(* PLC project Water_Reserve_Control, Desconocido Sin nombre 1 *)
(* stored: creationDateTime 2024-11-13T10:20:43, modificationDateTime 2024-11-13T13:10:53 *)

PROGRAM Water_Control
  VAR
    Pool_Low_Level_Sensor AT %IX0.0 : BOOL;  (* Pools Level Sensor signal of min level. Zero indicates that level is under the minimun *)
    Tank_High_Level_Sensor AT %IX0.1 : BOOL;  (* Tank Level Sensor of miax level. State "1" indicates maximun level *)
    Water_Pump AT %QX0.0 : BOOL;  (* Pump state control output. High value turns on the motor *)
    Tank_Low_Level_Sensor AT %IX0.2 : BOOL;  (* Tank Level Sensor of min level. Zero indicates that level is under the minimun *)
    Automatic_Manual_Switch AT %IX0.3 : BOOL;  (* Automatic/Manual selector. State "0" is Manual mode and "1" Automatic mode *)
    Stop_Button AT %IX0.4 : BOOL;  (* Stop Push Button. If changes its value to "1" indicates stop de pump *)
    Start_Button AT %IX0.5 : BOOL;  (* Start Push Button. If changes its value to "1" indicates start de pump *)
  END_VAR

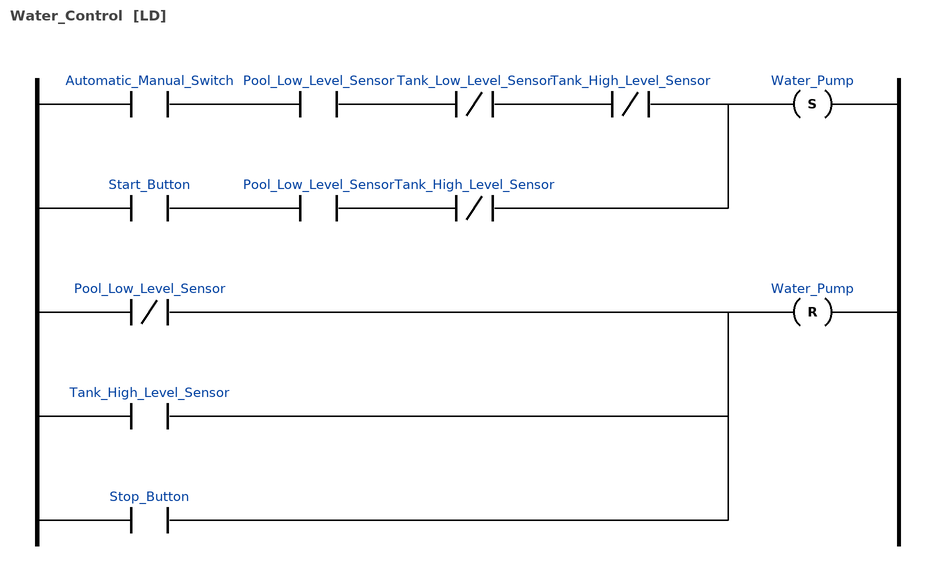
(* LD diagram, written out as Structured Text *)
IF Automatic_Manual_Switch AND Pool_Low_Level_Sensor AND NOT Tank_Low_Level_Sensor AND NOT Tank_High_Level_Sensor OR Start_Button AND Pool_Low_Level_Sensor AND NOT Tank_High_Level_Sensor THEN Water_Pump := TRUE; END_IF;
IF NOT Pool_Low_Level_Sensor OR Stop_Button OR Tank_High_Level_Sensor THEN Water_Pump := FALSE; END_IF;
END_PROGRAM

CONFIGURATION Config0
  RESOURCE Res0 ON PLC
    TASK task0(INTERVAL := T#20ms, PRIORITY := 0);
    PROGRAM instance0 WITH task0 : Water_Control;
  END_RESOURCE
END_CONFIGURATION
